# EPICS StreamDevice protocol: apps/dcPowerApp/Db/magflow.proto
#
#  MAGFLOW protocol definitions
#
Terminator = CR;
LockTimeout = 5000;
ReplyTimeout = 200;
ReadTimeout = 200;
WriteTimeout = 200;

get { out "\$1"; wait 50; in "%f"; }
